TYPE (* A Structure with 1 BOOL *)
  (* Version 1.0, 2024-02-21, Franz Höpfinger, HR Agrartechnik GmbH *)
  PACKAGE logiBUS::utils::conversion::types;
  IMPORT eclipse4diac::core::TypeHash;
  ST01X : STRUCT
    X_00 : BOOL; (* BIT 00 *)
  END_STRUCT;
END_TYPE
